FUNCTION_BLOCK StringBuilder255
VAR
	_Value : T_MaxString;
END_VAR

METHOD Append : REFERENCE TO StringBuilder255
VAR_INPUT
	value : T_MaxString;
END_VAR
Append REF= THIS^;

_Value := CONCAT(_Value, value);
END_METHOD

METHOD Clear : REFERENCE TO StringBuilder255
Clear REF= THIS^;

_Value := '';
END_METHOD

METHOD GetString : T_MaxString
GetString := _Value;
END_METHOD

PROPERTY IsEmpty : BOOL
GET
IsEmpty := Length = 0;
END_GET
END_PROPERTY

{attribute 'monitoring' := 'call'}
PROPERTY Length : DINT
GET
Length := LEN(_Value);
END_GET
END_PROPERTY

{attribute 'monitoring' := 'call'}
PROPERTY Value : T_MaxString
GET
Value := _Value;
END_GET
END_PROPERTY

END_FUNCTION_BLOCK

(* stored: Version 1.1.0.1
   POU StringBuilder255: Id {b6b3672a-e798-4798-8505-28948b4a51c2}, SpecialFunc None
   Method Append: Id {7f696451-9508-4294-997f-c551e4ac0594}
   Method Clear: Id {1edd4649-c2f3-4a46-85d1-e292ca0d812e}
   Method GetString: Id {b5dc5e56-10cd-471b-8d60-87863a4a2968}
   Property IsEmpty: Id {da104aa9-6c57-467c-8bb4-fd60c903a0ed}
   Get Get: Id {37dfe591-a83e-4a8a-ad72-8bf366367ede}
   Property Length: Id {d00c72c0-0b26-4fdd-bf24-d85486af71fa}
   Get Get: Id {7572048f-91f8-4c1a-9b4c-0ea4f7664396}
   Property Value: Id {d7164e58-869b-4ff5-8ffe-01fb4a8f62c6}
   Get Get: Id {72adfa88-ef38-4be2-93bb-16cf974a1295} *)
